// TIA Portal project "FactoryIO_Template_S7-1200_V16_V16" (V16)
// Vorlageprojekt für das Buch mit Zielsystem S7-1200

(* hardware
DEVICE "S7-1200-Station_1"  S7-1200 Station
   slot 0: "Baugruppenträger_0"  Rack  V1.0
   slot 1: "PLC_1"  CPU 1211C DC/DC/DC  6ES7 211-1AE40-0XB0  V4.1
*)

// ===== PLC "PLC_1"  CPU 1211C DC/DC/DC =====

VAR_GLOBAL   // PLC tag table "Standard-Variablentabelle"
   "green conveyor" AT %A0.0 : Bool;
   "start" AT %E0.0 : Bool;
   "Tag_3" AT %E0.1 : Bool;
   "Tag_4" AT %I10.0 : Bool;
   "Tag_5" AT %Q10.0 : Bool;
   "Tag_6" AT %I10.1 : Bool;
   "stop" AT %I0.2 : Bool;
   "x" AT %M0.0 : Bool;
   "middle conveyor" AT %Q0.1 : Bool;
   "blue conveyor" AT %Q0.2 : Bool;
   "diffuse sensor 2" AT %I0.3 : Bool;
   "diffuse sensor 1" AT %I0.4 : Bool;
   "diffuse sensor 4" AT %I0.5 : Bool;
   "diffuse sensor 5" AT %I0.6 : Bool;
   "Tag_1" AT %M0.2 : Bool;
   "c1(1)" AT %M0.3 : Bool;
   "diffuse sensor 3" AT %I0.7 : Bool;
   "pusher" AT %Q0.3 : Bool;
   "diffuse sensor 6" AT %I1.0 : Bool;
   "Tag_2" AT %M0.4 : Bool;
   "c2(1)" AT %M0.5 : Bool;
   "middle 2m" AT %Q0.4 : Bool;
   "y" AT %M0.6 : Bool;
   "Tag_7" AT %M1.0 : Bool;
   "z" AT %M1.1 : Bool;
   "Tag_8" AT %M1.2 : Bool;
   "Tag_9" AT %M2.0 : Bool;
   "Tag_10" AT %M2.1 : Bool;
   "Tag_11" AT %M2.2 : Bool;
   "Tag_12" AT %M3.0 : Bool;
   "Tag_13" AT %M3.1 : Bool;
END_VAR

// folder: System blocks/Program resources

DATA_BLOCK "C"   // DB2
{ S7_Optimized_Access := 'TRUE' }
AUTHOR : Simatic
FAMILY : IEC
NAME : CNTR
VERSION : 1.0
// stored: InstanceOfName IEC_COUNTER
"IEC_COUNTER"
BEGIN
END_DATA_BLOCK

DATA_BLOCK "C2"   // DB4
{ S7_Optimized_Access := 'TRUE' }
AUTHOR : Simatic
FAMILY : IEC
NAME : CNTR
VERSION : 1.0
// stored: InstanceOfName IEC_COUNTER
"IEC_COUNTER"
BEGIN
END_DATA_BLOCK

// folder: (top level)

FUNCTION "MHJ-PLC-Lab-Function-S71200" : Void   // FC9000, SCL
{ S7_Optimized_Access := 'TRUE' }
VERSION : 0.1
   VAR_TEMP
      rdTimeReturn : Int;
      outputTime : DTL;
      SyncVal : Byte;
      forVal : Int;
      forVal_2 : Int;
      Value : Byte;
   END_VAR
   VAR CONSTANT
      CompVal : Byte := 16#34;
      Value_01 : Byte := 16#11;
      Value_01_DW : DWord := 16#A165_D992;
      Value_02_DW : DWord := 16#58BE_4401;
   END_VAR
BEGIN

   #Value:=PEEK(area := 16#82,
        dbNumber := 0,
        byteOffset := 511);
   #Value := #Value + 1;

   POKE(area := 16#82,
        dbNumber := 0,
        byteOffset := 511,
        value := #Value);

   POKE(area:=16#81,
        dbNumber:=0,
        byteOffset:=1016,
        value:=#Value_01_DW);
   POKE(area := 16#81,
        dbNumber := 0,
        byteOffset := 1020,
        value := #Value_02_DW);

   POKE(area := 16#81,
        dbNumber := 0,
        byteOffset := 511,
        value := B#16#00);

   FOR #forVal := 0 TO 120 DO
       FOR #forVal_2:=0 TO 10 DO
           #rdTimeReturn:=RD_SYS_T(#outputTime);
           #rdTimeReturn := WR_SYS_T(#outputTime);
           #rdTimeReturn := RD_SYS_T(#outputTime);
           #rdTimeReturn := WR_SYS_T(#outputTime);
       END_FOR;
       #SyncVal:= PEEK(area := 16#81,
                      dbNumber := 0,
                      byteOffset := 511);
       IF #SyncVal = #CompVal THEN
          GOTO M_1;
       END_IF;
   END_FOR;
   RETURN;

   M_1:
   POKE(area := 16#81,
        dbNumber := 0,
        byteOffset := 511,
        value := B#16#0);
END_FUNCTION

ORGANIZATION_BLOCK "Main"   // OB1, LAD, ProgramCycle
TITLE = "Main Program Sweep (Cycle)"
{ S7_Optimized_Access := 'TRUE' }
VERSION : 0.1
   VAR_INPUT
      Initial_Call : Bool;   // Initial call of this OB
      Remanence : Bool;   // =True, if remanent data are available
   END_VAR
   VAR_TEMP   // added for the SCL form of the ladder/FBD networks
      _w1 : Bool;
      _w2 : Bool;
      _w3 : Bool;
      _w4 : Bool;
   END_VAR
BEGIN

REGION Network 1: Konnektierungsbaustein für PLC-Lab
   // Im Netzwerk 1 wird der Konnektierungsbaustein für PLC-Lab aufgerufen.
   // Dieser Aufruf darf nicht entfernt werden!
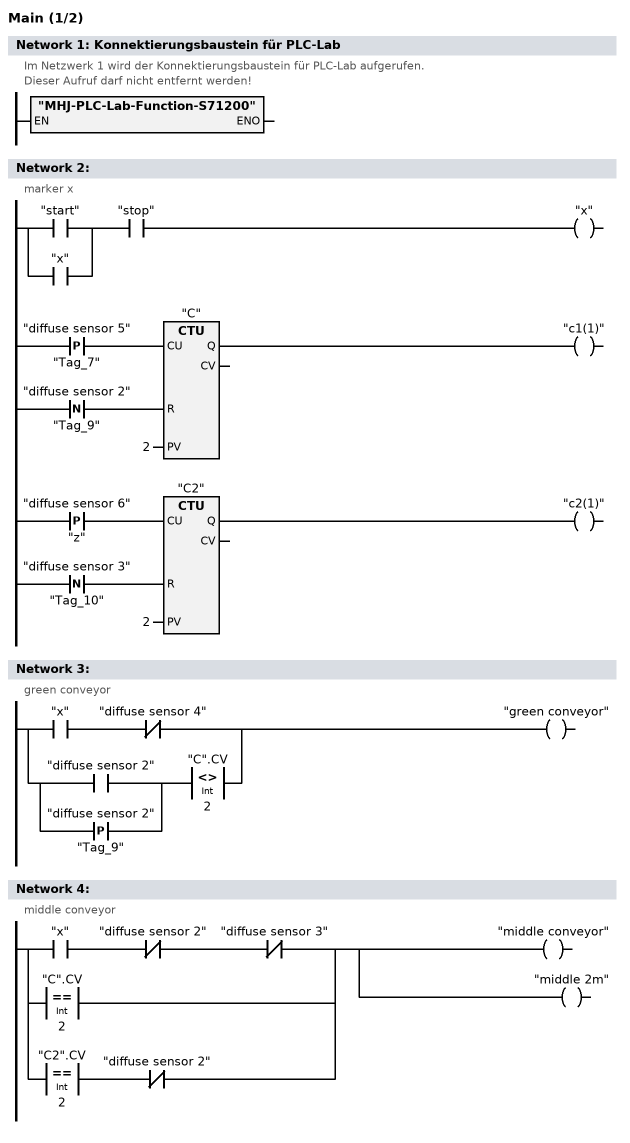
   RUNG wire#powerrail
      "MHJ-PLC-Lab-Function-S71200"()
   END_RUNG
   // the same network as SCL:
   "MHJ-PLC-Lab-Function-S71200"();
END_REGION

REGION Network 2
   // marker x
   "x" := ("start" OR "x") AND "stop";
   #_w1 := "diffuse sensor 5" AND NOT "Tag_7";   // rising edge of "diffuse sensor 5"
   "Tag_7" := "diffuse sensor 5";
   #_w2 := NOT "diffuse sensor 2" AND "Tag_9";   // falling edge of "diffuse sensor 2"
   "Tag_9" := "diffuse sensor 2";
   "C".CTU(CU := #_w1, R := #_w2, PV := 2);
   "c1(1)" := "C".Q;
   #_w3 := "diffuse sensor 6" AND NOT "z";   // rising edge of "diffuse sensor 6"
   "z" := "diffuse sensor 6";
   #_w4 := NOT "diffuse sensor 3" AND "Tag_10";   // falling edge of "diffuse sensor 3"
   "Tag_10" := "diffuse sensor 3";
   "C2".CTU(CU := #_w3, R := #_w4, PV := 2);
   "c2(1)" := "C2".Q;
END_REGION

REGION Network 3
   // green conveyor
   RUNG wire#powerrail
      Contact( "x" )
      I_Contact( "diffuse sensor 4" )
      wire#w1
      Coil( "green conveyor" )
   END_RUNG
   RUNG wire#powerrail
      Contact( "diffuse sensor 2" )
      wire#w2
      { S7_Templates := "SrcType := Int" } NE_Contact(in1 := "C".CV, in2 := 2)
   END_RUNG wire#w1
   RUNG wire#powerrail
      P_Contact(operand := "diffuse sensor 2", bit := "Tag_9")
   END_RUNG wire#w2
   // the same network as SCL:
   #_w1 := "diffuse sensor 2" AND NOT "Tag_9";   // rising edge of "diffuse sensor 2"
   "Tag_9" := "diffuse sensor 2";
   "green conveyor" := ("x" AND NOT "diffuse sensor 4") OR (("diffuse sensor 2" OR #_w1) AND ("C".CV <> 2));
END_REGION

REGION Network 4
   // middle conveyor
   RUNG wire#powerrail
      Contact( "x" )
      I_Contact( "diffuse sensor 2" )
      I_Contact( "diffuse sensor 3" )
      wire#w1
      Coil( "middle conveyor" )
   END_RUNG
   RUNG wire#powerrail
      { S7_Templates := "SrcType := Int" } EQ_Contact(in1 := "C".CV, in2 := 2)
   END_RUNG wire#w1
   RUNG wire#powerrail
      { S7_Templates := "SrcType := Int" } EQ_Contact(in1 := "C2".CV, in2 := 2)
      I_Contact( "diffuse sensor 2" )
   END_RUNG wire#w1
   RUNG wire#w1
      Coil( "middle 2m" )
   END_RUNG
   // the same network as SCL:
   "middle conveyor" := ("x" AND NOT "diffuse sensor 2" AND NOT "diffuse sensor 3") OR ("C".CV = 2) OR (("C2".CV = 2) AND NOT "diffuse sensor 2");
   "middle 2m" := "middle conveyor";
END_REGION

REGION Network 5
   // Blue conveyor
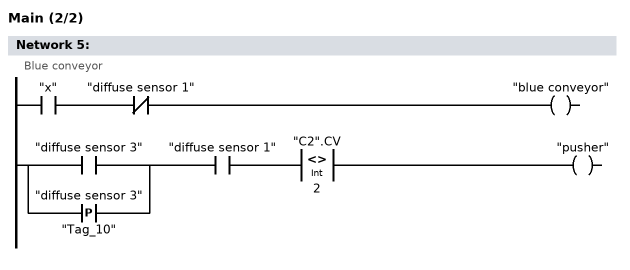
   RUNG wire#powerrail
      Contact( "x" )
      I_Contact( "diffuse sensor 1" )
      Coil( "blue conveyor" )
   END_RUNG
   RUNG wire#powerrail
      Contact( "diffuse sensor 3" )
      wire#w1
      Contact( "diffuse sensor 1" )
      { S7_Templates := "SrcType := Int" } NE_Contact(in1 := "C2".CV, in2 := 2)
      Coil( "pusher" )
   END_RUNG
   RUNG wire#powerrail
      P_Contact(operand := "diffuse sensor 3", bit := "Tag_10")
   END_RUNG wire#w1
   // the same network as SCL:
   "blue conveyor" := "x" AND NOT "diffuse sensor 1";
   #_w1 := "diffuse sensor 3" AND NOT "Tag_10";   // rising edge of "diffuse sensor 3"
   "Tag_10" := "diffuse sensor 3";
   "pusher" := ("diffuse sensor 3" OR #_w1) AND "diffuse sensor 1" AND ("C2".CV <> 2);
END_REGION
END_ORGANIZATION_BLOCK